FUNCTION TryConvert_WORD_TO_TOD : BOOL
VAR_INPUT
	in : WORD;
	out : REFERENCE TO TOD;
END_VAR

out := WORD_TO_TOD(in);
TryConvert_WORD_TO_TOD := TRUE;

END_FUNCTION

(* stored: Version 1.1.0.1, ProductVersion 3.1.4024.12
   POU TryConvert_WORD_TO_TOD: Id {18146614-db52-48b2-86a3-ff503a4f0188}, SpecialFunc None *)
